KUKA KRL program: ProfileWallDist.src, ProfileWallDist.dat

--- ProfileWallDist.src ---
&ACCESS RV2
&REL 8
DEFFCT REAL ProfileWallDist(eProfile:IN,eDim:IN,iWall:IN)
   DECL E_ProfileType eProfile
   DECL E_Dimension eDim
   DECL INT iWall
   DECL REAL rWallDist

   SWITCH eDim
      CASE #Y
         rWallDist = WallDistY(eProfile,iWall)
      CASE #Z
         rWallDist = WallDistZ(eProfile,iWall)
      DEFAULT
         HALT
   ENDSWITCH

   RETURN rWallDist

ENDFCT

;FOLD WallDistY()
   DEFFCT REAL WallDistY(eProfile:IN,iWall:IN)
      DECL E_ProfileType eProfile
      DECL INT iWall
      DECL REAL rWallDist

      SWITCH eProfile
         CASE #Leaf75
            rWallDist = rLeafY75[iWall]
         CASE #Leaf90
            rWallDist = rLeafY90[iWall]
         CASE #Frame75
            rWallDist = rFrameY75[iWall]
         CASE #Frame90
            rWallDist = rFrameY90[iWall]
         DEFAULT
            HALT
      ENDSWITCH

      RETURN rWallDist

   ENDFCT

;ENDFOLD

;FOLD WallDistZ()
   DEFFCT REAL WallDistZ(eProfile:IN,iWall:IN)
      DECL E_ProfileType eProfile
      DECL INT iWall
      DECL REAL rWallDist

      SWITCH eProfile
         CASE #Leaf75
            rWallDist = rLeafZ75[iWall]
         CASE #Leaf90
            rWallDist = rLeafZ90[iWall]
         CASE #Frame75
            rWallDist = rFrameZ75[iWall]
         CASE #Frame90
            rWallDist = rFrameZ90[iWall]
         CASE #Threshold90
            rWallDist = rThresholdZ90[iWall]
         DEFAULT
            HALT
      ENDSWITCH

      RETURN rWallDist

   ENDFCT

;ENDFOLD

--- ProfileWallDist.dat ---
&ACCESS RV2
&REL 8
DEFDAT ProfileWallDist

   ;Leaf 75
   DECL CONST REAL rLeafY75[4]
   rLeafY75[1] = 71.5
   rLeafY75[2] = 43.2
   rLeafY75[3] = 7.5
   rLeafY75[4] = 2.5
   DECL CONST REAL rLeafZ75[2]
   rLeafZ75[1] = 50.6
   rLeafZ75[2] = 2.5

   ;Leaf 90
   DECL CONST REAL rLeafY90[4]
   rLeafY90[1] = 85.7
   rLeafY90[2] = 68.5
   rLeafY90[3] = 32.5
   rLeafY90[4] = 3.0
   DECL CONST REAL rLeafZ90[2]
   rLeafZ90[1] = 48.8
   rLeafZ90[2] = 2.8

   ;Frame 75
   DECL CONST REAL rFrameY75[4]
   rFrameY75[1] = 75.8
   rFrameY75[2] = 45.0
   rFrameY75[3] = 9.5
   rFrameY75[4] = 2.8
   DECL CONST REAL rFrameZ75[2]
   rFrameZ75[1] = 45.5
   rFrameZ75[2] = 7.5

   ;Frame 90
   DECL CONST REAL rFrameY90[4]
   rFrameY90[1] = 90.8
   rFrameY90[2] = 59.3
   rFrameY90[3] = 23.4
   rFrameY90[4] = 2.6
   DECL CONST REAL rFrameZ90[2]
   rFrameZ90[1] = 52.7
   rFrameZ90[2] = 7.4

   ;Threshold 90
   DECL CONST REAL rThresholdZ90[2]
   rThresholdZ90[1] = 19.0
   rThresholdZ90[2] = 4.0

ENDDAT
